{attribute 'linkalways'} 
{attribute 'no_explicit_call' := 'This FB is a CLASS and must be accessed using methods or properties'}
{attribute 'enable_dynamic_creation'}
FUNCTION_BLOCK Node_F_VN_ContourCenterOfMass EXTENDS VisionNode
VAR
    ipContour : _ITcVnContainer;
    aCenterOfMass : _TcVnPoint2_LREAL;
    hrPrev : _HRESULT(S_OK);
	hresult : _HRESULT(S_OK);
END_VAR

METHOD PUBLIC  Clone : I_Node
VAR
	pNode : POINTER TO Node_F_VN_ContourCenterOfMass;
END_VAR
pNode := __NEW(Node_F_VN_ContourCenterOfMass);
Clone := pNode^;
END_METHOD

METHOD FB_init : BOOL
VAR_INPUT
	bInitRetains : BOOL; // if TRUE, the retain variables are initialized (warm start / cold start)
	bInCopyCode : BOOL;  // if TRUE, the instance afterwards gets moved into the copy code (online change)
END_VAR
AddInput('ipContour', ipContour);
AddInput('hrPrev', hrPrev);
AddOutput('aCenterOfMass', aCenterOfMass);
AddOutput('hresult',hresult);
END_METHOD

METHOD PROTECTED OnExecute
hresult.Value := F_VN_ContourCenterOfMass(
	ipContour := ipContour.Value,
    aCenterOfMass := aCenterOfMass.Value,
	hrPrev:= hrPrev.Value);
END_METHOD

METHOD PUBLIC PreExecutionCheck
VAR_INPUT
	Check : I_PreExecutionChecks;
END_VAR
Check.IsTrue(ipContour.IsValid, 'ipContour must be a valid container');
Check.IsTrue((ipContour.IsType(TC_GLOBAL_CONST_LIST.ContainerType_Vector_TcVnPoint2_DINT) OR
              ipContour.IsType(TC_GLOBAL_CONST_LIST.ContainerType_Vector_TcVnPoint2_REAL)),
              'ipContour contains incorrect type');
END_METHOD

END_FUNCTION_BLOCK

(* stored: Version 1.1.0.1, ProductVersion 3.1.4026.13
   POU Node_F_VN_ContourCenterOfMass: Id {e66c383f-2ee5-06f4-3079-22d2e7936d73}, SpecialFunc None
   Folder Constructor: Id {c07f3a9d-2295-0e07-0d0e-e3f7fc77b70c}
   Method Clone: Id {a3f286ed-5475-09f6-2984-1f59b5aa4fad}
   Method FB_init: Id {e60a1d9f-4047-0788-35dc-02a9e0ed8aba}
   Method OnExecute: Id {af414c20-9c1f-0e55-2750-a95f39e26c4a}
   Method PreExecutionCheck: Id {d420a0e7-600e-0d82-34bb-9d454a47add1} *)
